// LS Electric XG5000 project: 63_2_연습
// PLC NewPLC
// module base 0 slot 0: 입출력 모듈:XBC-DR20S (DC 24V 입력 12점, 릴레이 출력 8점)

PROGRAM NewProgram (task: 스캔 프로그램)

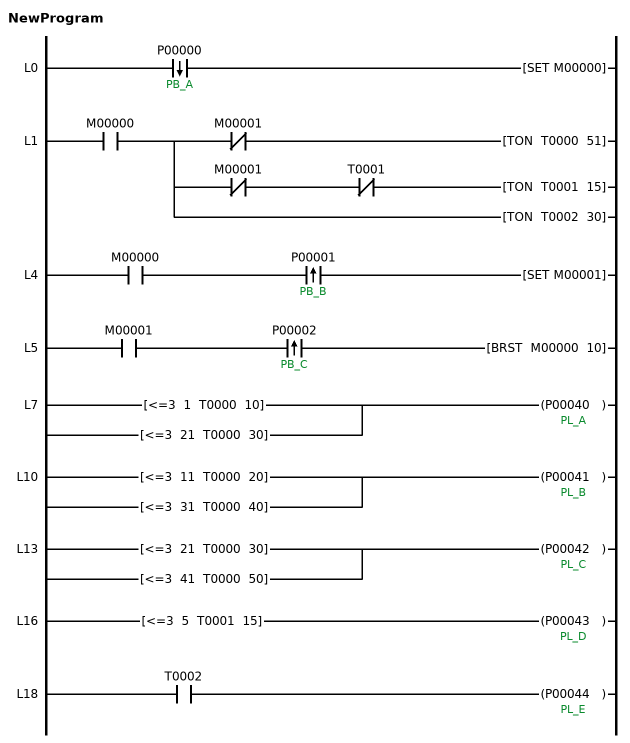
; L0
LOADN     P00000	// PB_A
SET       M00000
; L1
LOAD      M00000
MPUSH
AND NOT   M00001
TON       T0000 51
MLOAD
AND NOT   M00001
AND NOT   T0001
TON       T0001 15
MPOP
TON       T0002 30
; L4
LOAD      M00000
ANDP      P00001	// PB_B
SET       M00001
; L5
LOAD      M00001
ANDP      P00002	// PB_C
BRST      M00000 10
; L7
LOAD<=3   1 T0000 10
OR<=3     21 T0000 30
OUT       P00040	// PL_A
; L10
LOAD<=3   11 T0000 20
OR<=3     31 T0000 40
OUT       P00041	// PL_B
; L13
LOAD<=3   21 T0000 30
OR<=3     41 T0000 50
OUT       P00042	// PL_C
; L16
LOAD<=3   5 T0001 15
OUT       P00043	// PL_D
; L18
LOAD      T0002
OUT       P00044	// PL_E